(* Logix 5000 project; controller AplicacionAFEbancoDePruebas vendor 1 type 14 code 149 rev 33.12; software revision 33.01 *)

TASK MainTask (continuous, watchdog 500 ms) : MainProgram

MODULES
   Local : vendor 1 type 14 code 149 (Compact 0, rev 33.12)
      Discrete_IO : Embedded (Compact 1, rev 3.1, Output RPI 20 ms)
      PLC : 1769-L32E Ethernet Port (Ethernet 192.168.2.131, rev 20.1)
         PLC_Controller : vendor 1 type 14 code 77 (CompactLogixL32EController 0, rev 20.1, $d20f6a59$ RPI 20 ms, $b1273c18$ RPI 20 ms, $a621ca3b$ RPI 20 ms)
      VSD_AFE : vendor 1 type 143 code 8336 (Ethernet 192.168.2.50, rev 6.5, Output RPI 20 ms)
           VSD_AFE:O.LogicCommand_Stop   // Comando de Parada
           VSD_AFE:O.LogicCommand_Start   // Comando de Arranque
          : vendor 1 type 143 code 161 (RhinoBP 10, rev 1.1)
          : vendor 1 type 143 code 416 (RhinoBP 5, rev 1.8)
          : vendor 1 type 143 code 675 (RhinoBP 13, rev 1.1)
          : vendor 1 type 143 code 416 (RhinoBP 4, rev 1.8)
          : vendor 1 type 143 code 2724 (RhinoBP 14, rev 1.1)
          : vendor 1 type 143 code 4770 (RhinoBP 12, rev 1.1)
END_MODULES

TYPE Dinagrama :   // Estructura para el dinagrama
STRUCT
   vPotencia : REAL[500];   // captura del vector de potencia
   vCarga : REAL[500];   // captura del vector de carga
   vPosicion : REAL[500];   // captura del vector posicion
   vProximetro : DINT[500];   // captura del vector del proximetro
   NumeroMuestras : INT;
   enabled : BOOL;
   captura : BOOL;   // Flag que indica la captura del sistema
   resetVector : BOOL;   // Flag para darle Reset al vector de posición y carga
   vEmptyREAL : REAL[500];
   vEmptyINT : DINT[500];
END_STRUCT
END_TYPE

TYPE LSW :   // Drive - Logic Status Word
STRUCT
   Faulted : BOOL;
   Warning : BOOL;
   RunForward : BOOL;
   RunReverse : BOOL;
   Ready : BOOL;
   RemoteRef : BOOL;
   RemoteCrtl : BOOL;
   AtSpeed : BOOL;
END_STRUCT
END_TYPE

TYPE SWC :
STRUCT
   Dinagrama : Dinagrama;
   VSD : VSD;
   entradasDigitales : INT;   // Entradas Digitales
   salidasDigitales : INT;   // Salidas Digitales
   entradasAnalogas : REAL[4];   // Entradas Analogas del PLC
   salidasAnalogas : REAL[4];
END_STRUCT
END_TYPE

TYPE VSD :   // VSD
STRUCT
   VSD_O : AB:PowerFlex755T_E_31635488:O:0;
   VSD_I : AB:PowerFlex755T_E_2B0A69C5:I:0;
END_STRUCT
END_TYPE

VAR_GLOBAL   (* controller tags *)
   SRP_Displacement_Actual : REAL := 68.22777;   // Variable de Simulacion PLC DC de Desplazamiento
   SRP_Load_Actual : REAL := 10.401504;   // Variable de simulacion PLC DC de Carga
   SRP_SimActualStroke : DINT;   // Variable Simulación de PLC Variador DC
   SWC : SWC := (Dinagrama.vPotencia[0] := 0.0018305705, Dinagrama.vPotencia[1] := 0.0017222156, Dinagrama.vPotencia[2] := 0.0016868035, Dinagrama.vPotencia[4] := 0.0016790881, Dinagrama.vPotencia[5] := 0.0017240789, Dinagrama.vPotencia[6] := 0.0017701827, Dinagrama.vPotencia[7] := 0.0018443047, Dinagrama.vPotencia[8] := 0.0018918252, Dinagrama.vPotencia[9] := 0.0019517487, Dinagrama.vPotencia[10] := 0.001982275, Dinagrama.vPotencia[12] := 0.0019949286, Dinagrama.vPotencia[14] := 0.0019226995, Dinagrama.vPotencia[15] := 0.0018463905, Dinagrama.vPotencia[16] := 0.0017900213, Dinagrama.vPotencia[18] := 0.0016542743, Dinagrama.vPotencia[19] := 0.001637371, Dinagrama.vPotencia[21] := 0.0017060273, Dinagrama.vPotencia[22] := 0.0017597966, Dinagrama.vPotencia[24] := 0.0018860088, Dinagrama.vPotencia[29] := 0.0019709691, Dinagrama.vPotencia[35] := 0.0016295084, Dinagrama.vPotencia[36] := 0.0016458338, Dinagrama.vPotencia[37] := 0.0017049119, Dinagrama.vPotencia[41] := 0.0019425809, Dinagrama.vPotencia[44] := 0.001972656, Dinagrama.vPotencia[47] := 0.0018182971, Dinagrama.vPotencia[49] := 0.0016925418, Dinagrama.vPotencia[53] := 0.0017570421, Dinagrama.vPotencia[55] := 0.0018721677, Dinagrama.vPotencia[66] := 0.0016643361, Dinagrama.vPotencia[68] := 0.0017211302, Dinagrama.vPotencia[70] := 0.0018310223, Dinagrama.vPotencia[72] := 0.0019449221, Dinagrama.vPotencia[74] := 0.0020018201, Dinagrama.vPotencia[76] := 0.00197123, Dinagrama.vPotencia[78] := 0.0018768503, Dinagrama.vPotencia[81] := 0.0016752455, Dinagrama.vPotencia[84] := 0.0017242664, Dinagrama.vPotencia[86] := 0.0018486312, Dinagrama.vPotencia[89] := 0.0019866459, Dinagrama.vPotencia[90] := 0.0020152421, Dinagrama.vPotencia[93] := 0.0019546899, Dinagrama.vPotencia[96] := 0.0017026957, Dinagrama.vPotencia[98] := 0.0016592251, Dinagrama.vPotencia[100] := 0.0017287023, Dinagrama.vPotencia[102] := 0.0018590746, Dinagrama.vPotencia[106] := 0.001997631, Dinagrama.vPotencia[108] := 0.001958732, Dinagrama.vPotencia[110] := 0.0018284139, Dinagrama.vPotencia[112] := 0.0016919352, Dinagrama.vPotencia[114] := 0.0016496999, Dinagrama.vPotencia[116] := 0.0017337679, Dinagrama.vPotencia[120] := 0.0019674972, Dinagrama.vPotencia[122] := 0.0019990792, Dinagrama.vPotencia[123] := 0.001992557, Dinagrama.vPotencia[124] := 0.0019616408, Dinagrama.vPotencia[126] := 0.0018534678, Dinagrama.vPotencia[127] := 0.0017874483, Dinagrama.vPotencia[129] := 0.0016443202, Dinagrama.vPotencia[132] := 0.0017402298,
        Dinagrama.vPotencia[134] := 0.0018691482, Dinagrama.vPotencia[136] := 0.001968309, Dinagrama.vPotencia[138] := 0.001996729, Dinagrama.vPotencia[139] := 0.0019830258, Dinagrama.vPotencia[142] := 0.0018053686, Dinagrama.vPotencia[143] := 0.0018053686, Dinagrama.vPotencia[144] := 0.0020029054, Dinagrama.vPotencia[145] := 0.0019953735, Dinagrama.vPotencia[147] := 0.001955511, Dinagrama.vPotencia[148] := 0.0019137838, Dinagrama.vPotencia[149] := 0.0037706406, Dinagrama.vPotencia[151] := 0.003613952, Dinagrama.vPotencia[154] := 0.0016774976, Dinagrama.vPotencia[155] := 0.001643918, Dinagrama.vPotencia[156] := 0.001637348, Dinagrama.vPotencia[158] := 0.0016542862, Dinagrama.vPotencia[161] := 0.0017273742, Dinagrama.vPotencia[163] := 0.0018007061, Dinagrama.vPotencia[164] := 0.0018473662, Dinagrama.vPotencia[165] := 0.0018695425, Dinagrama.vPotencia[166] := 0.0019162475, Dinagrama.vPotencia[168] := 0.0034027533, Dinagrama.vPotencia[169] := 0.0019702422, Dinagrama.vPotencia[170] := 0.0019748174, Dinagrama.vPotencia[171] := 0.0019841003, Dinagrama.vPotencia[172] := 0.0034300725, Dinagrama.vPotencia[173] := 0.0019587537, Dinagrama.vPotencia[175] := 0.0033207624, Dinagrama.vPotencia[176] := 0.0018908933, Dinagrama.vPotencia[178] := 0.0017995888, Dinagrama.vPotencia[179] := 0.003059388, Dinagrama.vPotencia[180] := 0.0016968154, Dinagrama.vPotencia[182] := 0.0032600476, Dinagrama.vPotencia[185] := 0.001639651, Dinagrama.vPotencia[187] := 0.001691746, Dinagrama.vPotencia[189] := 0.0030624089, Dinagrama.vPotencia[193] := 0.0019071687, Dinagrama.vPotencia[194] := 0.0038546922, Dinagrama.vPotencia[195] := 0.0019580075, Dinagrama.vPotencia[196] := 0.00341182, Dinagrama.vPotencia[197] := 0.003982586, Dinagrama.vPotencia[199] := 0.0019969982, Dinagrama.vPotencia[200] := 0.0019861378, Dinagrama.vPotencia[201] := 0.0019679056, Dinagrama.vPotencia[202] := 0.001933599, Dinagrama.vPotencia[203] := 0.0019164722, Dinagrama.vPotencia[204] := 0.0018507714, Dinagrama.vPotencia[206] := 0.0030501464, Dinagrama.vPotencia[207] := 0.00172522, Dinagrama.vPotencia[209] := 0.001645268, Dinagrama.vPotencia[210] := 0.0028384142, Dinagrama.vPotencia[211] := 0.0016229607, Dinagrama.vPotencia[213] := 0.0028661871, Dinagrama.vPotencia[216] := 0.0017448035, Dinagrama.vPotencia[218] := 0.0018252019, Dinagrama.vPotencia[220] := 0.0038026192, Dinagrama.vPotencia[223] := 0.0019714264, Dinagrama.vPotencia[224] := 0.0019905828, Dinagrama.vPotencia[225] := 0.001993408, Dinagrama.vPotencia[226] := 0.00391313,
        Dinagrama.vPotencia[228] := 0.003708509, Dinagrama.vPotencia[229] := 0.0017909358, Dinagrama.vPotencia[230] := 0.0017025609, Dinagrama.vPotencia[232] := 0.0033112175, Dinagrama.vPotencia[233] := 0.0016824467, Dinagrama.vPotencia[234] := 0.0017266382, Dinagrama.vPotencia[235] := 0.0017758736, Dinagrama.vPotencia[240] := 0.0016576217, Dinagrama.vPotencia[241] := 0.001661227, Dinagrama.vPotencia[242] := 0.0044334494, Dinagrama.vPotencia[243] := 0.003408804, Dinagrama.vPotencia[245] := 0.003530516, Dinagrama.vCarga[0] := 9.794512, Dinagrama.vCarga[1] := 9.714645, Dinagrama.vCarga[2] := 9.698671, Dinagrama.vCarga[3] := 9.858406, Dinagrama.vCarga[4] := 9.858406, Dinagrama.vCarga[5] := 9.762565, Dinagrama.vCarga[6] := 9.682698, Dinagrama.vCarga[7] := 9.570884, Dinagrama.vCarga[8] := 9.666724, Dinagrama.vCarga[9] := 10.177875, Dinagrama.vCarga[10] := 10.177875, Dinagrama.vCarga[11] := 10.449424, Dinagrama.vCarga[12] := 10.593185, Dinagrama.vCarga[13] := 10.832787, Dinagrama.vCarga[14] := 10.976549, Dinagrama.vCarga[15] := 11.389862, Dinagrama.vCarga[16] := 11.389862, Dinagrama.vCarga[17] := 11.477716, Dinagrama.vCarga[18] := 11.591527, Dinagrama.vCarga[19] := 11.783209, Dinagrama.vCarga[20] := 11.851096, Dinagrama.vCarga[21] := 11.99885, Dinagrama.vCarga[22] := 11.825139, Dinagrama.vCarga[23] := 11.563573, Dinagrama.vCarga[24] := 11.214154, Dinagrama.vCarga[25] := 11.040442, Dinagrama.vCarga[26] := 10.848761, Dinagrama.vCarga[27] := 10.625132, Dinagrama.vCarga[28] := 10.465398, Dinagrama.vCarga[29] := 10.321636, Dinagrama.vCarga[30] := 10.193849, Dinagrama.vCarga[31] := 10.018141, Dinagrama.vCarga[32] := 9.842432, Dinagrama.vCarga[33] := 9.682698, Dinagrama.vCarga[34] := 9.586857, Dinagrama.vCarga[35] := 9.826459, Dinagrama.vCarga[36] := 10.050088, Dinagrama.vCarga[37] := 10.113981, Dinagrama.vCarga[38] := 10.241769, Dinagrama.vCarga[39] := 10.401504, Dinagrama.vCarga[40] := 10.417477, Dinagrama.vCarga[41] := 10.401504, Dinagrama.vCarga[42] := 10.513318, Dinagrama.vCarga[43] := 10.545265, Dinagrama.vCarga[44] := 10.449424, Dinagrama.vCarga[45] := 10.609159, Dinagrama.vCarga[46] := 10.75292, Dinagrama.vCarga[47] := 10.529291,
        Dinagrama.vCarga[48] := 10.209822, Dinagrama.vCarga[49] := 9.986194, Dinagrama.vCarga[50] := 9.890353, Dinagrama.vCarga[51] := 9.650751, Dinagrama.vCarga[52] := 9.395175, Dinagrama.vCarga[53] := 9.411149, Dinagrama.vCarga[54] := 9.379202, Dinagrama.vCarga[55] := 9.155573, Dinagrama.vCarga[56] := 9.011812, Dinagrama.vCarga[57] := 9.123626, Dinagrama.vCarga[58] := 8.995839, Dinagrama.vCarga[59] := 8.788184, Dinagrama.vCarga[60] := 9.043759, Dinagrama.vCarga[61] := 9.379202, Dinagrama.vCarga[62] := 9.522963, Dinagrama.vCarga[63] := 9.60283, Dinagrama.vCarga[64] := 9.842432, Dinagrama.vCarga[65] := 9.842432, Dinagrama.vCarga[66] := 9.97022, Dinagrama.vCarga[67] := 10.002167, Dinagrama.vCarga[68] := 9.954247, Dinagrama.vCarga[69] := 10.034114, Dinagrama.vCarga[70] := 9.986194, Dinagrama.vCarga[71] := 9.986194, Dinagrama.vCarga[72] := 10.098008, Dinagrama.vCarga[73] := 10.193849, Dinagrama.vCarga[74] := 9.618804, Dinagrama.vCarga[75] := 9.538937, Dinagrama.vCarga[76] := 9.55491, Dinagrama.vCarga[77] := 9.55491, Dinagrama.vCarga[78] := 9.331282, Dinagrama.vCarga[79] := 9.171547, Dinagrama.vCarga[80] := 9.315308, Dinagrama.vCarga[81] := 9.123626, Dinagrama.vCarga[82] := 9.123626, Dinagrama.vCarga[83] := 9.18752, Dinagrama.vCarga[84] := 9.331282, Dinagrama.vCarga[85] := 9.18752, Dinagrama.vCarga[86] := 9.155573, Dinagrama.vCarga[87] := 9.522963, Dinagrama.vCarga[88] := 9.778539, Dinagrama.vCarga[89] := 9.682698, Dinagrama.vCarga[90] := 9.714645, Dinagrama.vCarga[91] := 9.906326, Dinagrama.vCarga[92] := 9.874379, Dinagrama.vCarga[93] := 9.634777, Dinagrama.vCarga[94] := 9.634777, Dinagrama.vCarga[95] := 9.666724, Dinagrama.vCarga[96] := 9.411149, Dinagrama.vCarga[97] := 9.203494, Dinagrama.vCarga[98] := 9.09168, Dinagrama.vCarga[99] := 8.820131, Dinagrama.vCarga[100] := 8.3569, Dinagrama.vCarga[101] := 7.957564, Dinagrama.vCarga[102] := 7.89367, Dinagrama.vCarga[103] := 7.765882, Dinagrama.vCarga[104] := 7.462386, Dinagrama.vCarga[105] := 7.270704, Dinagrama.vCarga[106] := 7.302651, Dinagrama.vCarga[107] := 7.11097,
        Dinagrama.vCarga[108] := 6.759554, Dinagrama.vCarga[109] := 6.599819, Dinagrama.vCarga[110] := 6.839421, Dinagrama.vCarga[111] := 7.031103, Dinagrama.vCarga[112] := 7.254731, Dinagrama.vCarga[113] := 7.622121, Dinagrama.vCarga[114] := 7.925617, Dinagrama.vCarga[115] := 7.909643, Dinagrama.vCarga[116] := 7.909643, Dinagrama.vCarga[117] := 8.245086, Dinagrama.vCarga[118] := 8.3569, Dinagrama.vCarga[119] := 8.324953, Dinagrama.vCarga[120] := 8.596502, Dinagrama.vCarga[121] := 8.804157, Dinagrama.vCarga[122] := 8.788184, Dinagrama.vCarga[123] := 8.788184, Dinagrama.vCarga[124] := 8.756237, Dinagrama.vCarga[125] := 8.420794, Dinagrama.vCarga[126] := 8.340927, Dinagrama.vCarga[127] := 8.484688, Dinagrama.vCarga[128] := 8.388847, Dinagrama.vCarga[129] := 8.452741, Dinagrama.vCarga[130] := 8.596502, Dinagrama.vCarga[131] := 8.500661, Dinagrama.vCarga[132] := 8.484688, Dinagrama.vCarga[133] := 8.484688, Dinagrama.vCarga[134] := 8.564555, Dinagrama.vCarga[135] := 8.564555, Dinagrama.vCarga[136] := 8.804157, Dinagrama.vCarga[137] := 9.043759, Dinagrama.vCarga[138] := 9.043759, Dinagrama.vCarga[139] := 9.267388, Dinagrama.vCarga[140] := 9.331282, Dinagrama.vCarga[141] := 9.299335, Dinagrama.vCarga[142] := 9.682698, Dinagrama.vCarga[143] := 9.682698, Dinagrama.vPosicion[0] := 0.330105, Dinagrama.vPosicion[1] := 0.799962, Dinagrama.vPosicion[2] := 1.393695, Dinagrama.vPosicion[3] := 2.117669, Dinagrama.vPosicion[4] := 2.117669, Dinagrama.vPosicion[5] := 2.974185, Dinagrama.vPosicion[6] := 3.96401, Dinagrama.vPosicion[7] := 6.2659, Dinagrama.vPosicion[8] := 7.553576, Dinagrama.vPosicion[9] := 8.91896, Dinagrama.vPosicion[10] := 8.91896, Dinagrama.vPosicion[11] := 10.358983, Dinagrama.vPosicion[12] := 11.886531, Dinagrama.vPosicion[13] := 13.500606, Dinagrama.vPosicion[14] := 15.167234, Dinagrama.vPosicion[15] := 18.670801, Dinagrama.vPosicion[16] := 18.670801, Dinagrama.vPosicion[17] := 20.497496, Dinagrama.vPosicion[18] := 22.359915, Dinagrama.vPosicion[19] := 24.276115, Dinagrama.vPosicion[20] := 26.231995, Dinagrama.vPosicion[21] := 28.230639, Dinagrama.vPosicion[22] := 30.26319, Dinagrama.vPosicion[23] := 32.348446,
        Dinagrama.vPosicion[24] := 34.475838, Dinagrama.vPosicion[25] := 36.630318, Dinagrama.vPosicion[26] := 38.818886, Dinagrama.vPosicion[27] := 41.046406, Dinagrama.vPosicion[28] := 43.30216, Dinagrama.vPosicion[29] := 45.59054, Dinagrama.vPosicion[30] := 47.925312, Dinagrama.vPosicion[31] := 50.300934, Dinagrama.vPosicion[32] := 52.57733, Dinagrama.vPosicion[33] := 54.853752, Dinagrama.vPosicion[34] := 57.161697, Dinagrama.vPosicion[35] := 59.435463, Dinagrama.vPosicion[36] := 61.651955, Dinagrama.vPosicion[37] := 63.858036, Dinagrama.vPosicion[38] := 66.06483, Dinagrama.vPosicion[39] := 68.22777, Dinagrama.vPosicion[40] := 70.327156, Dinagrama.vPosicion[41] := 72.39657, Dinagrama.vPosicion[42] := 74.43364, Dinagrama.vPosicion[43] := 76.41475, Dinagrama.vPosicion[44] := 78.31727, Dinagrama.vPosicion[45] := 80.16558, Dinagrama.vPosicion[46] := 81.96299, Dinagrama.vPosicion[47] := 83.7108, Dinagrama.vPosicion[48] := 85.39305, Dinagrama.vPosicion[49] := 86.980385, Dinagrama.vPosicion[50] := 88.4902, Dinagrama.vPosicion[51] := 89.93009, Dinagrama.vPosicion[52] := 91.27383, Dinagrama.vPosicion[53] := 92.51773, Dinagrama.vPosicion[54] := 93.67952, Dinagrama.vPosicion[55] := 94.75152, Dinagrama.vPosicion[56] := 95.7108, Dinagrama.vPosicion[57] := 96.58106, Dinagrama.vPosicion[58] := 97.35993, Dinagrama.vPosicion[59] := 98.024086, Dinagrama.vPosicion[60] := 98.59063, Dinagrama.vPosicion[61] := 99.06094, Dinagrama.vPosicion[62] := 99.44078, Dinagrama.vPosicion[63] := 99.71841, Dinagrama.vPosicion[64] := 99.902794, Dinagrama.vPosicion[65] := 99.902794, Dinagrama.vPosicion[66] := 99.99385, Dinagrama.vPosicion[67] := 99.91777, Dinagrama.vPosicion[68] := 99.73818, Dinagrama.vPosicion[69] := 99.471176, Dinagrama.vPosicion[70] := 99.1364, Dinagrama.vPosicion[71] := 99.1364, Dinagrama.vPosicion[72] := 98.72924, Dinagrama.vPosicion[73] := 98.26827, Dinagrama.vPosicion[74] := 97.14606, Dinagrama.vPosicion[75] := 97.14606, Dinagrama.vPosicion[76] := 95.795845, Dinagrama.vPosicion[77] := 95.795845, Dinagrama.vPosicion[78] := 95.004196, Dinagrama.vPosicion[79] := 94.16693, Dinagrama.vPosicion[80] := 92.36308, Dinagrama.vPosicion[81] := 91.377556, Dinagrama.vPosicion[82] := 91.377556, Dinagrama.vPosicion[83] := 90.37801,
        Dinagrama.vPosicion[84] := 89.32036, Dinagrama.vPosicion[85] := 88.20336, Dinagrama.vPosicion[86] := 87.044815, Dinagrama.vPosicion[87] := 85.84824, Dinagrama.vPosicion[88] := 84.59012, Dinagrama.vPosicion[89] := 83.28975, Dinagrama.vPosicion[90] := 81.95589, Dinagrama.vPosicion[91] := 80.55808, Dinagrama.vPosicion[92] := 79.11205, Dinagrama.vPosicion[93] := 77.63775, Dinagrama.vPosicion[94] := 76.10894, Dinagrama.vPosicion[95] := 74.51687, Dinagrama.vPosicion[96] := 72.905495, Dinagrama.vPosicion[97] := 71.262856, Dinagrama.vPosicion[98] := 69.54499, Dinagrama.vPosicion[99] := 67.80591, Dinagrama.vPosicion[100] := 66.05848, Dinagrama.vPosicion[101] := 64.23761, Dinagrama.vPosicion[102] := 62.366978, Dinagrama.vPosicion[103] := 60.49874, Dinagrama.vPosicion[104] := 58.589725, Dinagrama.vPosicion[105] := 56.612167, Dinagrama.vPosicion[106] := 54.624504, Dinagrama.vPosicion[107] := 52.632183, Dinagrama.vPosicion[108] := 50.586884, Dinagrama.vPosicion[109] := 48.494823, Dinagrama.vPosicion[110] := 46.39611, Dinagrama.vPosicion[111] := 44.280315, Dinagrama.vPosicion[112] := 42.1344, Dinagrama.vPosicion[113] := 39.97316, Dinagrama.vPosicion[114] := 37.810795, Dinagrama.vPosicion[115] := 35.634483, Dinagrama.vPosicion[116] := 33.423225, Dinagrama.vPosicion[117] := 31.23504, Dinagrama.vPosicion[118] := 29.075682, Dinagrama.vPosicion[119] := 26.898933, Dinagrama.vPosicion[120] := 24.743301, Dinagrama.vPosicion[121] := 22.634195, Dinagrama.vPosicion[122] := 20.581553, Dinagrama.vPosicion[123] := 18.588135, Dinagrama.vPosicion[124] := 16.676949, Dinagrama.vPosicion[125] := 14.84577, Dinagrama.vPosicion[126] := 13.085015, Dinagrama.vPosicion[127] := 11.417382, Dinagrama.vPosicion[128] := 9.842795, Dinagrama.vPosicion[129] := 8.365165, Dinagrama.vPosicion[130] := 6.990245, Dinagrama.vPosicion[131] := 5.721944, Dinagrama.vPosicion[132] := 4.565173, Dinagrama.vPosicion[133] := 4.565173, Dinagrama.vPosicion[134] := 2.64918, Dinagrama.vPosicion[135] := 2.64918, Dinagrama.vPosicion[136] := 1.232986, Dinagrama.vPosicion[137] := 0.727498, Dinagrama.vPosicion[138] := 0.727498, Dinagrama.vPosicion[139] := 0.354476, Dinagrama.vPosicion[140] := 0.1153, Dinagrama.vPosicion[142] := 0.059576, Dinagrama.vPosicion[143] := 0.059576, Dinagrama.vProximetro[0] := 1,
        Dinagrama.vProximetro[1] := 1, Dinagrama.vProximetro[2] := 1, Dinagrama.vProximetro[3] := 1, Dinagrama.vProximetro[4] := 1, Dinagrama.vProximetro[5] := 1, Dinagrama.vProximetro[6] := 1, Dinagrama.vProximetro[245] := 1, Dinagrama.vProximetro[247] := 1, Dinagrama.vProximetro[248] := 1, Dinagrama.vProximetro[249] := 1, Dinagrama.vProximetro[250] := 1, Dinagrama.vProximetro[251] := 1, Dinagrama.vProximetro[252] := 1, Dinagrama.vProximetro[253] := 1, Dinagrama.vProximetro[254] := 1, Dinagrama.vProximetro[255] := 1, Dinagrama.vProximetro[256] := 1, Dinagrama.vProximetro[257] := 1, Dinagrama.vProximetro[258] := 1, Dinagrama.vProximetro[494] := 1, Dinagrama.vProximetro[495] := 1, Dinagrama.vProximetro[496] := 1, Dinagrama.vProximetro[497] := 1, Dinagrama.vProximetro[498] := 1, Dinagrama.vProximetro[499] := 1, Dinagrama.NumeroMuestras := 143, Dinagrama.enabled := 1, VSD.VSD_O.P10_VRefAStpt := 0.6316, VSD.VSD_I.DriveStatus := 2#1010_0000_0010_0001_0000_0101_0000_1111, VSD.VSD_I.DriveStatus_Ready := 1, VSD.VSD_I.DriveStatus_Active := 1, VSD.VSD_I.DriveStatus_CommandDir := 1, VSD.VSD_I.DriveStatus_ActualDir := 1, VSD.VSD_I.DriveStatus_AtSpeed := 1, VSD.VSD_I.DriveStatus_SpdRefBit0 := 1, VSD.VSD_I.DriveStatus_Running := 1, VSD.VSD_I.DriveStatus_SpeedMode := 1, VSD.VSD_I.DriveStatus_EnableOn := 1, VSD.VSD_I.DriveStatus_Regen := 1, VSD.VSD_I.Feedback := 0.6316, VSD.VSD_I.P10_VRefCommanded := 0.63159996, VSD.VSD_I.P12_M0CurrentFdbkW := 0.2856468, VSD.VSD_I.P10_OutputVoltage := 9.078274, VSD.VSD_I.P10_OutputPower := 0.0020036423, VSD.VSD_I.P13_PowerFactor := -0.07546366, VSD.VSD_I.DCBusVolts := 704.5499, VSD.VSD_I.P10_HeatsnkTemp := 23.186409, VSD.VSD_I.ElapsedRunTime := 19.989, VSD.VSD_I.LastFaultCode := 14136, VSD.VSD_I.ElapsedkWH := -11143, VSD.VSD_I.P10_OutputCurrent := 0.1438037, entradasDigitales := 3, entradasAnalogas[0] := -1.7e-44, entradasAnalogas[1] := -9.176336e+29, entradasAnalogas[2] := 3.8693e-41, entradasAnalogas[3] := 6.66079e-40, salidasAnalogas[0] := 1.e-45, salidasAnalogas[1] := 6.e-45, salidasAnalogas[2] := 4.e-45);
        .Dinagrama.enabled   // Habilitar Adquision
END_VAR

PROGRAM MainProgram   (* main routine R000_MainRoutine *)
VAR
   Captura : BOOL;
   contadorAux : ALIAS FOR counter[0].ACC;
   counter : COUNTER[10];
   Enabled : BOOL;
   Flag : BOOL;
   habilitar : DINT;
   myoneshot : BOOL[32] := ([1] := 1, [2] := 1);
        [0]   // oneshot toogle bot dinagrama
        [1]   // oneshor reset del ocntador
        [2]   // reset de la flag cuando se habilita y se deshabilita
   Proximetro_Virtual : ALIAS FOR SRP_SimActualStroke;
   SPM_Reference : REAL := 8.5;
   timer : TIMER[10] := ([0].PRE := 50);
        [0]   // Tiempo Muestreo
END_VAR

ROUTINE R000_MainRoutine   (* ladder *)
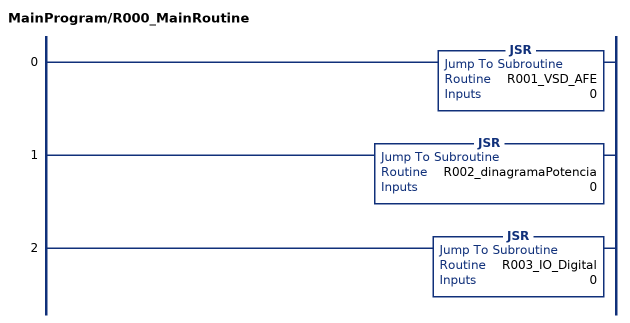
   0: JSR(R001_VSD_AFE,0);
   1: JSR(R002_dinagramaPotencia,0);
   2: JSR(R003_IO_Digital,0);
END_ROUTINE

ROUTINE R001_VSD_AFE   (* ladder *)
// Comandos Basicos de Operación de VSD AFE
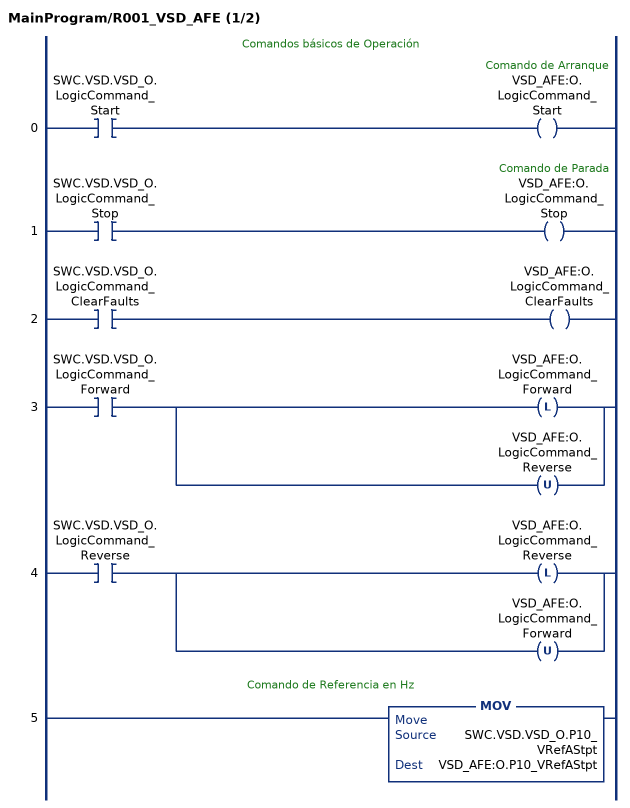
   // Comandos básicos de Operación
   0: XIC(SWC.VSD.VSD_O.LogicCommand_Start)OTE(VSD_AFE:O.LogicCommand_Start);
   1: XIC(SWC.VSD.VSD_O.LogicCommand_Stop)OTE(VSD_AFE:O.LogicCommand_Stop);
   2: XIC(SWC.VSD.VSD_O.LogicCommand_ClearFaults)OTE(VSD_AFE:O.LogicCommand_ClearFaults);
   3: XIC(SWC.VSD.VSD_O.LogicCommand_Forward)[OTL(VSD_AFE:O.LogicCommand_Forward) ,OTU(VSD_AFE:O.LogicCommand_Reverse) ];
   4: XIC(SWC.VSD.VSD_O.LogicCommand_Reverse)[OTL(VSD_AFE:O.LogicCommand_Reverse) ,OTU(VSD_AFE:O.LogicCommand_Forward) ];
   // Comando de Referencia en Hz
   5: MOV(SWC.VSD.VSD_O.P10_VRefAStpt,VSD_AFE:O.P10_VRefAStpt);
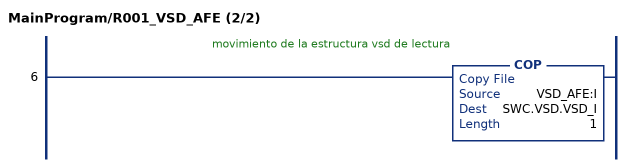
   // movimiento de la estructura vsd de lectura
   6: COP(VSD_AFE:I,SWC.VSD.VSD_I,1);
END_ROUTINE

ROUTINE R002_dinagramaPotencia   (* ladder *)
// Adquisión de los diferentes strokes para la captura del dinagrama de superficie
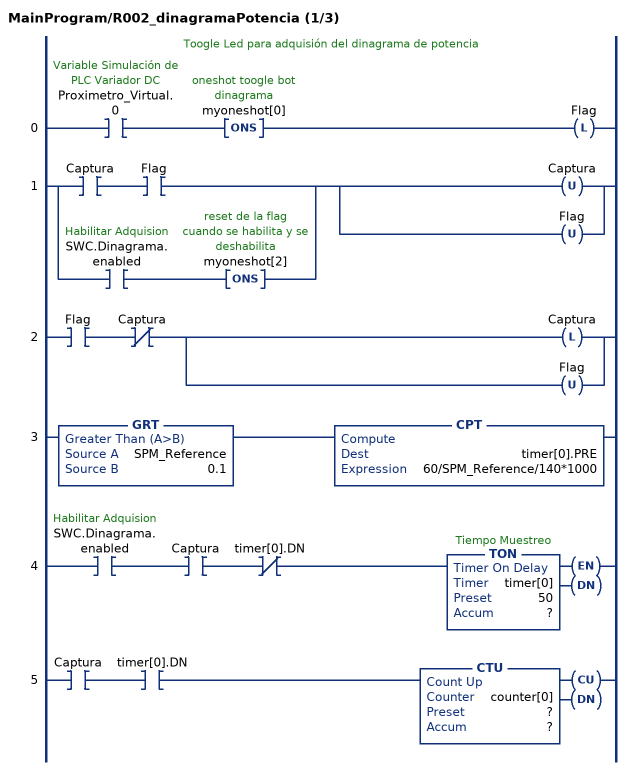
   // Toogle Led para adquisión del dinagrama de potencia
   0: XIC(Proximetro_Virtual.0)ONS(myoneshot[0])OTL(Flag);
   1: [XIC(Captura) XIC(Flag) ,XIC(SWC.Dinagrama.enabled) ONS(myoneshot[2]) ][OTU(Captura) ,OTU(Flag) ];
   2: XIC(Flag)XIO(Captura)[OTL(Captura) ,OTU(Flag) ];
   3: GRT(SPM_Reference,0.1)CPT(timer[0].PRE,60/SPM_Reference/140*1000);
   4: XIC(SWC.Dinagrama.enabled)XIC(Captura)XIO(timer[0].DN)TON(timer[0],?,?);
   5: XIC(Captura)XIC(timer[0].DN)CTU(counter[0],?,?);
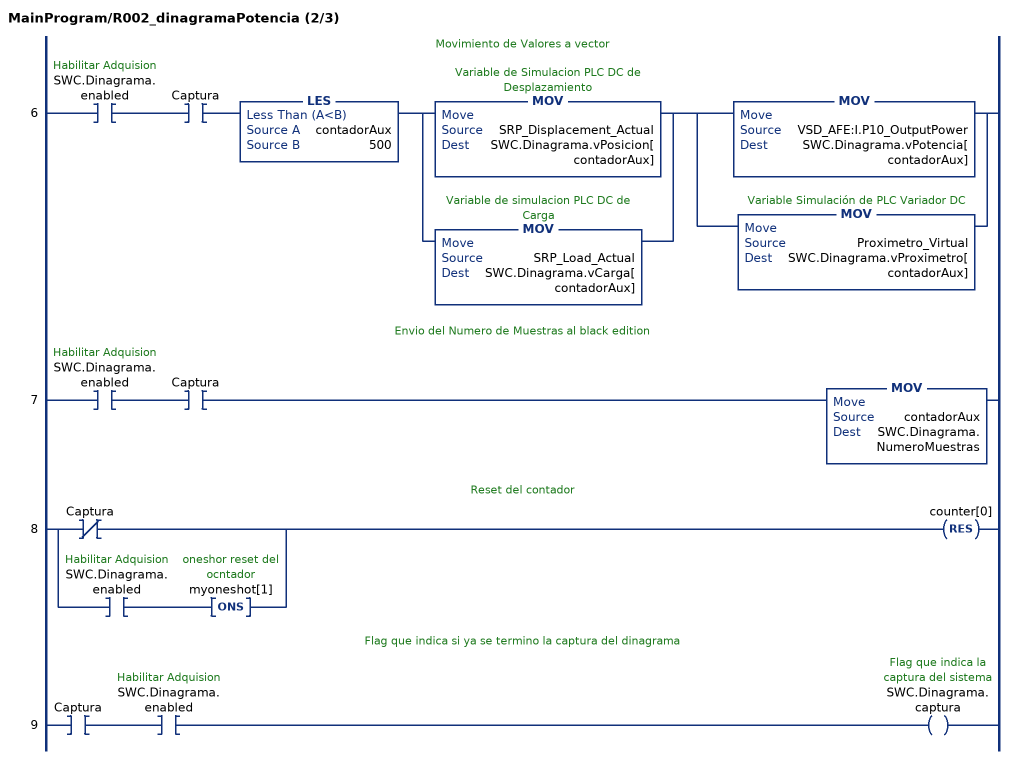
   // Movimiento de Valores a vector
   6: XIC(SWC.Dinagrama.enabled)XIC(Captura)LES(contadorAux,500)[MOV(SRP_Displacement_Actual,SWC.Dinagrama.vPosicion[contadorAux]) ,MOV(SRP_Load_Actual,SWC.Dinagrama.vCarga[contadorAux]) ][MOV(VSD_AFE:I.P10_OutputPower,SWC.Dinagrama.vPotencia[contadorAux]) ,MOV(Proximetro_Virtual,SWC.Dinagrama.vProximetro[contadorAux]) ];
   // Envio del Numero de Muestras al black edition
   7: XIC(SWC.Dinagrama.enabled)XIC(Captura)MOV(contadorAux,SWC.Dinagrama.NumeroMuestras);
   // Reset del contador
   8: [XIO(Captura) ,XIC(SWC.Dinagrama.enabled) ONS(myoneshot[1]) ]RES(counter[0]);
   // Flag que indica si ya se termino la captura del dinagrama
   9: XIC(Captura)XIC(SWC.Dinagrama.enabled)OTE(SWC.Dinagrama.captura);
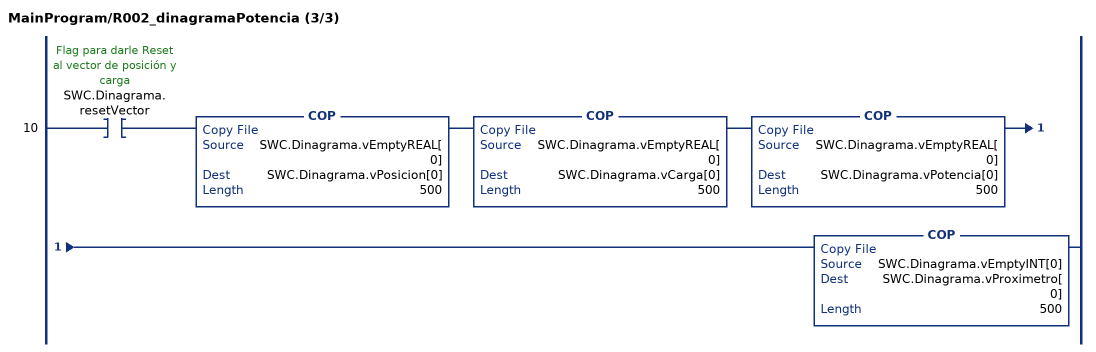
   10: XIC(SWC.Dinagrama.resetVector)COP(SWC.Dinagrama.vEmptyREAL[0],SWC.Dinagrama.vPosicion[0],500)COP(SWC.Dinagrama.vEmptyREAL[0],SWC.Dinagrama.vCarga[0],500)COP(SWC.Dinagrama.vEmptyREAL[0],SWC.Dinagrama.vPotencia[0],500)COP(SWC.Dinagrama.vEmptyINT[0],SWC.Dinagrama.vProximetro[0],500);
END_ROUTINE

ROUTINE R003_IO_Digital   (* ladder *)
// Entradas Digitales
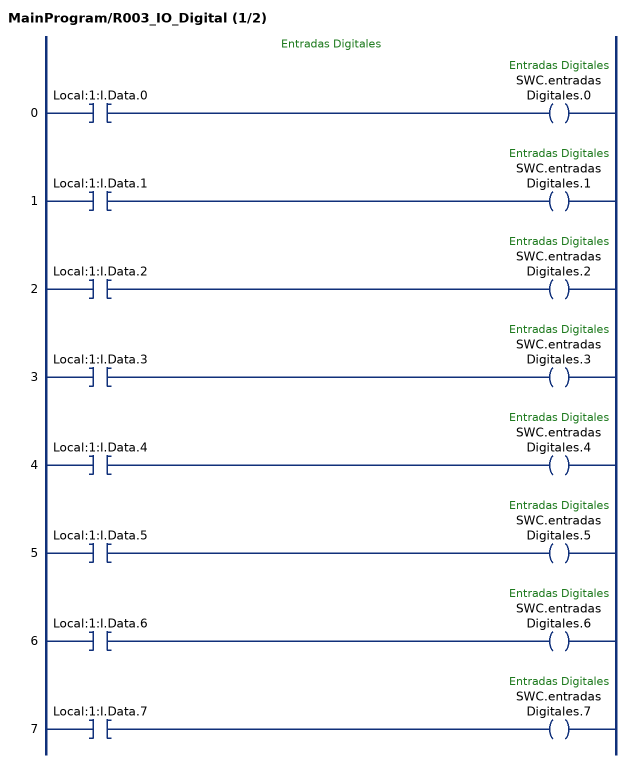
   // Entradas Digitales
   0: XIC(Local:1:I.Data.0)OTE(SWC.entradasDigitales.0);
   1: XIC(Local:1:I.Data.1)OTE(SWC.entradasDigitales.1);
   2: XIC(Local:1:I.Data.2)OTE(SWC.entradasDigitales.2);
   3: XIC(Local:1:I.Data.3)OTE(SWC.entradasDigitales.3);
   4: XIC(Local:1:I.Data.4)OTE(SWC.entradasDigitales.4);
   5: XIC(Local:1:I.Data.5)OTE(SWC.entradasDigitales.5);
   6: XIC(Local:1:I.Data.6)OTE(SWC.entradasDigitales.6);
   7: XIC(Local:1:I.Data.7)OTE(SWC.entradasDigitales.7);
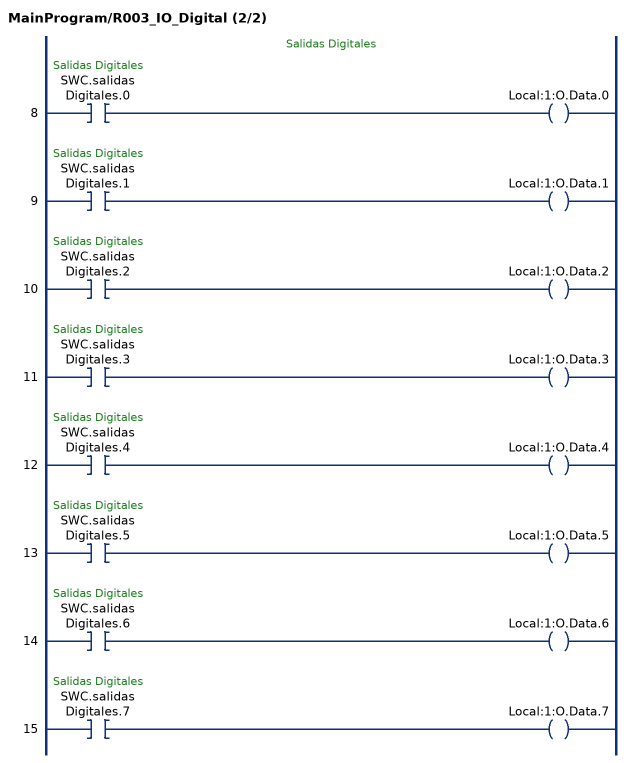
   // Salidas Digitales
   8: XIC(SWC.salidasDigitales.0)OTE(Local:1:O.Data.0);
   9: XIC(SWC.salidasDigitales.1)OTE(Local:1:O.Data.1);
   10: XIC(SWC.salidasDigitales.2)OTE(Local:1:O.Data.2);
   11: XIC(SWC.salidasDigitales.3)OTE(Local:1:O.Data.3);
   12: XIC(SWC.salidasDigitales.4)OTE(Local:1:O.Data.4);
   13: XIC(SWC.salidasDigitales.5)OTE(Local:1:O.Data.5);
   14: XIC(SWC.salidasDigitales.6)OTE(Local:1:O.Data.6);
   15: XIC(SWC.salidasDigitales.7)OTE(Local:1:O.Data.7);
END_ROUTINE
END_PROGRAM
